// TIA Portal V16 export
// export: Created 2023-03-29T11:03:36.1285041Z, ExportSetting WithDefaults, DisplayName Totally Integrated Automation Portal, DisplayVersion V16 Update 6, DisplayName TIA Portal Version Control Interface, DisplayVersion V16 Update 2, DisplayName TIA Portal Openness, DisplayVersion V16 Update 6, DisplayName STEP 7 Professional, DisplayVersion V16 Update 6, DisplayName STEP 7 Safety, DisplayVersion V16, DisplayName WinCC Advanced, DisplayVersion V16 Update 6
DATA_BLOCK "ERR_Enum"   // DB105
{ S7_Optimized_Access := 'TRUE' }
VERSION : 0.1
// stored: AutoNumber false, DBAccessibleFromOPCUA true, IsOnlyStoredInLoadMemory false, IsRetainMemResEnabled false, IsWriteProtectedInAS false, MemoryReserve 0
   VAR
      GetErrorID : Array[0..27] of Word;
      SoftwareError { S7_SetPoint := 'True'} : "stt_ERR_Enum_SoftwareError";
      OB80 : Array[0..5] of Byte;
   END_VAR
BEGIN
   GetErrorID[0] := 16#2503;
   GetErrorID[1] := 16#2520;
   GetErrorID[2] := 16#2522;
   GetErrorID[3] := 16#2523;
   GetErrorID[4] := 16#2524;
   GetErrorID[5] := 16#2525;
   GetErrorID[6] := 16#2528;
   GetErrorID[7] := 16#2529;
   GetErrorID[8] := 16#252C;
   GetErrorID[9] := 16#2530;
   GetErrorID[10] := 16#2533;
   GetErrorID[11] := 16#2538;
   GetErrorID[12] := 16#2539;
   GetErrorID[13] := 16#253A;
   GetErrorID[14] := 16#253C;
   GetErrorID[15] := 16#253D;
   GetErrorID[16] := 16#253E;
   GetErrorID[17] := 16#253F;
   GetErrorID[18] := 16#2550;
   GetErrorID[19] := 16#2551;
   GetErrorID[20] := 16#2575;
   GetErrorID[21] := 16#2576;
   GetErrorID[22] := 16#2577;
   GetErrorID[23] := 16#25A0;
   GetErrorID[24] := 16#25A1;
   GetErrorID[25] := 16#25A2;
   GetErrorID[26] := 16#2942;
   GetErrorID[27] := 16#2943;
END_DATA_BLOCK
